(*

.. <legal notes>

legal notes
=================
| SPDX-FileCopyrightText: © 2025 Oleksandr Tiutyk <trofimich@gmail.com>
| SPDX-License-Identifier: LGPL-3.0-only
| For details check: LGPL-3.0-only_

.. _LGPL-3.0-only: https://www.gnu.org/licenses/lgpl-3.0.en.html

.. </legal notes>

*)

PROGRAM GenericValueHelper

METHOD CheckIsNull : BOOL
VAR_INPUT
	value : GENERIC_VALUE;
END_VAR
CheckIsNull := value.Address = 0 OR_ELSE value.Size = 0 OR_ELSE value.TypeClass = __SYSTEM.TYPE_CLASS.TYPE_NONE;
END_METHOD

{attribute 'monitoring' := 'call'}
PROPERTY NamespaceName : STRING
GET
NamespaceName := CurrentNamespace.Name;
END_GET
END_PROPERTY

END_PROGRAM

(* stored: Version 1.1.0.1
   POU GenericValueHelper: Id {632192a8-a1bb-419c-8eaa-096811803723}, SpecialFunc None
   Method CheckIsNull: Id {a4b85fbd-3ab9-4498-9490-7c058ad28188}
   Property NamespaceName: Id {86abee5b-3405-4bc7-a70a-27f1e1674f57}
   Get Get: Id {242c0548-b017-4d3b-96bc-df4db08b14ee} *)
